FUNCTION_BLOCK fbModTCP_Core IMPLEMENTS iModbusTcpCore
VAR_INPUT
	stTimeStruct : stAircomTimeStruct;																						// Time struct for data ack
END_VAR
VAR_OUTPUT
END_VAR
VAR
	fbModbusTCP 					: FB_MBReadWriteRegs;																	// Main function for ModbusTCP
	arCommQue						: ARRAY[0..GVL_ModbusTCP_Constants.iQueLimit] OF stModTcpQue;							// Que for core
	arModTcpCommandHist				: ARRAY[0..GVL_ModbusTCP_Constants.iCommuniactionHistoryLimit]  OF stModTcpHist;		// Saving of prcesed command
	iWorkStep						: INT;																					// Workstep
	stCommToPerform					: stModTcpQue;																			// Block for process purpose
	iLastQue						: UINT;																					// Que for commands
	iActualQue						: UINT;																					// Actualy performed register of que
	iHistory						: UINT;																					// History record
	rCommunicationTime				: REAL;																					// Time of communication
	fbCommTimeON					: R_TRIG;																				// Start of modbus block - Rise Edge
	fbCommTimeOFF					: F_TRIG;																				// End of modbus block - Falling Edge
	fbErrorDetect					: R_TRIG;																				// Error detected status
	iErrorCalc						: INT;																					// Calculation of errors
	//Visu
	stHMI							: stModTcpCore_HmiData;																	// Data for HMI purpose
	rTimeForStatistic				: REAL;																					// Time variable for statistic calculation - per second
	iLastQueStat					: UINT;																					// Amount of data saved to que
	iActualQueStat					: UINT;																					// Amount od data procesed
	arVisuHist						: ARRAY[0..GVL_ModbusTCP_Constants.iCommuniactionHistoryLimit] OF STRING;				// Command History
	iAmoutOfPerformedCommunications	: DWORD;																				// Sum amount of performed data exchange - per second
	iAmoutOfErrors					: DWORD;																				// Sum amount of errsrs during data exchange - per second
	rTimeforMinuteStatitic			: REAL;																					// Time variable for statistic calculation - per minute
	iLastQueStatMinute				: UINT;																					// Sum amount of performed data exchange - per minute
	iActualQueStatMinute			: UINT;																					// Sum amount of errors during data exchange - per minute
	arErrorHistory					: ARRAY[0..GVL_ModbusTCP_Constants.iCommunicationErrorHistory] OF STRING;				// Data of errors during communicaiotn
	iErrorHistoryIdentifier			: UINT;																					// Calculation of error history
END_VAR

//Rdzeń komuniakcji ModbusTCP
//TO-DO
//Dodać możliwość node - wiele jednoczesnych pracesów
//Dodać możliwosć wymiany inforamcji w Coilach
//Poprawiać ewentualnie wystepujące błędy


ACT_Background();
//Main loop

CASE iWorkStep OF
	0: 		//Inicialization - Step 1
		iWorkStep := 5;

	5: 		//Inicialization - Step 2
		iWorkStep := 10;

	10: 	//Wait for next operaiton
		IF arCommQue[iActualQue].sMachineIndifiner <> '' AND NOT fbModbusTCP.bBusy THEN
			iWorkStep := 15;
		ELSIF NOT fbModbusTCP.bBusy THEN
			IF iActualQue >= GVL_ModbusTCP_Constants.iQueLimit-1 THEN
				iActualQue := 0;
			ELSE
				iActualQue := iActualQue + 1;
			END_IF
		END_IF
	15:		// Check next command
			iWorkStep := 20;
	20:		// Operation prepare - Rewrite for command to perform
		stCommToPerform	:= arCommQue[iActualQue];
		iWorkStep := 25;
	25:		//Clear Que - only one command
		MEMSET(destAddr:=ADR(arCommQue[iActualQue]),fillByte:=0,n:=SIZEOF(stModTcpQue));
		iWorkStep := 30;
		iAmoutOfPerformedCommunications := iAmoutOfPerformedCommunications + 1;
	30:		//Insert command to comm block
		fbModbusTCP.sIPAddr 			:=	stCommToPerform.sIpAdress;
		fbModbusTCP.nUnitID				:=	stCommToPerform.iUnitId;
		fbModbusTCP.nTCPPort			:=	stCommToPerform.iPort;
		fbModbusTCP.nMBReadAddr 		:= 	stCommToPerform.iRegisterReadStartAdress;
		fbModbusTCP.nMBWriteAddr 		:= 	stCommToPerform.iRegisterWriteStartAdress;
			// Dodać error w przypadku ilości rejestrów większych od iWriteRegisterLimit/2
		fbModbusTCP.nReadQuantity 		:=	stCommToPerform.wRegistersReadQuantity;
		fbModbusTCP.nWriteQuantity		:=	stCommToPerform.wRegistersWriteQuantity;
			//Source - Data tobe written in slave | Destination - Data to be read form slave
		fbModbusTCP.cbSrcLength 		:= SIZEOF(stCommToPerform.arRegisterWriteArray^);
		fbModbusTCP.pSrcAddr 			:= stCommToPerform.arRegisterWriteArray;
		fbModbusTCP.cbDestLength 		:= SIZEOF(stCommToPerform.arRegisterReadArray^);
		fbModbusTCP.pDestAddr 			:= stCommToPerform.arRegisterReadArray;
			//Check if history buffer is full - if yes start form 0
		IF iHistory >= GVL_ModbusTCP_Constants.iCommuniactionHistoryLimit THEN
			iHistory := 0;
		END_IF
		arModTcpCommandHist[iHistory].sIpAdress 			:= 	stCommToPerform.sIpAdress;
		arModTcpCommandHist[iHistory].iUnitId 				:=	stCommToPerform.iUnitId;
		arModTcpCommandHist[iHistory].iPort 				:=	stCommToPerform.iPort;
		arModTcpCommandHist[iHistory].sMachineIndifiner 	:= 	stCommToPerform.sMachineIndifiner;
		arModTcpCommandHist[iHistory].sTimeString 			:= 	stTimeStruct.sTimeString;
		arVisuHist[iHistory] := CONCAT(STR1:=arModTcpCommandHist[iHistory].sIpAdress ,STR2:=' | ');
		arVisuHist[iHistory] := CONCAT(STR1:=arVisuHist[iHistory] ,STR2:=arModTcpCommandHist[iHistory].sMachineIndifiner);
		arVisuHist[iHistory] := CONCAT(STR1:=arVisuHist[iHistory] ,STR2:=' | ');
		arVisuHist[iHistory] := CONCAT(STR1:=arVisuHist[iHistory] ,STR2:= arModTcpCommandHist[iHistory].sTimeString);
		arVisuHist[iHistory] := CONCAT(STR1:=arVisuHist[iHistory] ,STR2:=' | ');
		
		iWorkStep := 40;
	40:		// Data exchange start
		fbModbusTCP.bExecute := TRUE;
		IF fbModbusTCP.bBusy THEN
			fbModbusTCP.bExecute := FALSE;
			iWorkStep := 50;
		END_IF
	50: 	//Wait for not busy
		IF NOT fbModbusTCP.bBusy THEN
			iWorkStep := 10;
		END_IF

END_CASE

ACTION ACT_Background:
// Main function
fbModbusTCP();
//Error counting
fbErrorDetect(CLK:= fbModbusTCP.bError);
IF fbErrorDetect.Q THEN
	iErrorCalc := iErrorCalc + 1;
	iAmoutOfErrors := iAmoutOfErrors + 1;
	arErrorHistory[iErrorHistoryIdentifier] := CONCAT(STR1:= stCommToPerform.sMachineIndifiner,STR2:=' | ');
	arErrorHistory[iErrorHistoryIdentifier] := CONCAT(STR1:= arErrorHistory[iErrorHistoryIdentifier],STR2:=stCommToPerform.sIpAdress);
	arErrorHistory[iErrorHistoryIdentifier] := CONCAT(STR1:= arErrorHistory[iErrorHistoryIdentifier],STR2:=' | ');
	arErrorHistory[iErrorHistoryIdentifier] := CONCAT(STR1:= arErrorHistory[iErrorHistoryIdentifier],STR2:=LREAL_TO_FMTSTR(in:=rCommunicationTime,iPrecision:=3,bRound:= FALSE));
	arErrorHistory[iErrorHistoryIdentifier] := CONCAT(STR1:= arErrorHistory[iErrorHistoryIdentifier],STR2:=' | ');
	arErrorHistory[iErrorHistoryIdentifier] := CONCAT(STR1:= arErrorHistory[iErrorHistoryIdentifier],STR2:=UDINT_TO_STRING(fbModbusTCP.nErrId));
	iErrorHistoryIdentifier := iErrorHistoryIdentifier + 1;
END_IF
// Clear amount of errors
IF fbModbusTCP.cbRead <> 0 THEN
	iErrorCalc := 0;
END_IF

//Communication statistic
fbCommTimeON(CLK:= fbModbusTCP.bBusy);
fbCommTimeOFF(CLK:= fbModbusTCP.bBusy);
IF fbCommTimeON.Q THEN
	rCommunicationTime := 0;
END_IF
IF fbModbusTCP.bBusy THEN
	rCommunicationTime := rCommunicationTime + 0.01;
END_IF
IF fbCommTimeOFF.Q THEN
	arModTcpCommandHist[iHistory].rCommandTime := rCommunicationTime;
	arVisuHist[iHistory] := CONCAT(STR1:=arVisuHist[iHistory] ,STR2:=LREAL_TO_FMTSTR(in:=rCommunicationTime,iPrecision:=3,bRound:= FALSE));
	arVisuHist[iHistory] := CONCAT(STR1:=arVisuHist[iHistory] ,STR2:=' | ');
	arModTcpCommandHist[iHistory].nErrorId := fbModbusTCP.nErrId;
	arVisuHist[iHistory] := CONCAT(STR1:=arVisuHist[iHistory] ,STR2:=UDINT_TO_STRING(arModTcpCommandHist[iHistory].nErrorId));
	iHistory := iHistory + 1;
	iActualQueStat := iActualQueStat + 1;
END_IF

//HMI

stHMI.arVisuHist 						:= arVisuHist;
stHMI.arErrorHistory 					:= arErrorHistory;
stHMI.iActualQue 						:= iActualQue;
stHMI.iAmoutOfErrors 					:= iAmoutOfErrors;
stHMI.iAmoutOfPerformedCommunications 	:= iAmoutOfPerformedCommunications;
stHMI.iLastQue 							:= iLastQue;
stHMI.iMessagesPerMinute 				:= iActualQueStatMinute;
stHMI.iPullsPerrMinute					:= iLastQueStatMinute;

IF stHMI.bClearStatistic THEN
	iAmoutOfPerformedCommunications := 0;
	iAmoutOfErrors := 0;
	iActualQueStatMinute := 0;
	iLastQueStatMinute := 0;
	iErrorHistoryIdentifier := 0;
	iHistory := 0;
	stHMI.bClearStatistic := FALSE;
	MEMSET(destAddr:=ADR(arErrorHistory),fillByte:=0,n:= SIZEOF(arErrorHistory));
	MEMSET(destAddr:=ADR(arVisuHist),fillByte:=0,n:= SIZEOF(arVisuHist));
END_IF

IF rTimeForStatistic >= GVL_ModbusTCP_Constants.rTimeForSecondStatistic THEN
	stHMI.iMessagesPerSecond := iActualQueStat;
	stHMI.iPullsPerSecond	:= iLastQueStat;
	iActualQueStatMinute := iActualQueStatMinute + iActualQueStat;
	iLastQueStatMinute	:= iLastQueStatMinute + iLastQueStat;
	iLastQueStat 	:= 0;
	iActualQueStat	:= 0;
	rTimeForStatistic := 0;
END_IF

IF rTimeforMinuteStatitic >= GVL_ModbusTCP_Constants.rTimeForMinuteStatistic THEN
	iActualQueStatMinute := 0;
	iLastQueStatMinute := 0;
	rTimeforMinuteStatitic := 0;
END_IF

rTimeForStatistic := rTimeForStatistic + 0.01;
rTimeforMinuteStatitic := rTimeforMinuteStatitic + 0.01;

fbModbusTCP.tTimeout := GVL_ModbusTCP_Constants.tModbusCommunicationTimeOut;
END_ACTION

METHOD mAddToQue : nModbusTCP_CommandStatus;
VAR_INPUT
	stCommParams	: stModTcpQue;
END_VAR
VAR
END_VAR
IF stCommParams.sIpAdress <> '' AND stCommParams.iPort <> 0 AND stCommParams.sMachineIndifiner <> '' 
AND stCommParams.arRegisterReadArray <> 0 AND stCommParams.arRegisterWriteArray <> 0 AND stCommParams.wRegistersReadQuantity <> 0 AND stCommParams.wRegistersWriteQuantity <> 0
AND stCommParams.wRegistersReadQuantity <= 2*SIZEOF(stCommParams.arRegisterReadArray^) AND stCommParams.wRegistersWriteQuantity <= 2*SIZEOF(stCommParams.arRegisterWriteArray^) THEN
	//IF arCommQue[iLastQue].sMachineIndifiner = stCommParams.sMachineIndifiner THEN
		//mAddToQue := nModbusTCP_CommandStatus.nCommandAlreadyinQue_03;
	//ELSE
		IF iLastQue >= GVL_ModbusTCP_Constants.iQueLimit THEN
			iLastQue := 0;
		END_IF
		IF arCommQue[iLastQue].sMachineIndifiner <> '' THEN
			mAddToQue := nModbusTCP_CommandStatus.nRecordAllreadyInUse_04;
			iLastQue := iLastQue + 1;
			iLastQueStat := iLastQueStat + 1;
		ELSE
			arCommQue[iLastQue] := stCommParams;
			mAddToQue := nModbusTCP_CommandStatus.nCommandPerformed_01;
			iLastQue := iLastQue + 1;
			iLastQueStat := iLastQueStat + 1;
		END_IF
	//END_IF
ELSE
	mAddToQue := nModbusTCP_CommandStatus.nCommandWrongParams_02;
END_IF
END_METHOD

{attribute 'monitoring' := 'call'}
PROPERTY pError : BOOL
GET
pError := iErrorCalc >= GVL_ModbusTCP_Constants.iErrorLimit;
END_GET
END_PROPERTY

END_FUNCTION_BLOCK

(* stored: Version 1.1.0.1, ProductVersion 3.1.4024.13
   POU fbModTCP_Core: Id {1eebaeb0-68d5-4ffe-85ae-e4bdd94758f4}, SpecialFunc None
   Action ACT_Background: Id {3293cfc1-0622-4dd3-8ae2-5d0eb1a0ab74}
   Method mAddToQue: Id {6fcee0ac-971a-4c86-9aba-3116f2e46b99}
   Property pError: Id {362ccfd9-47cc-416e-ab04-599a1a60cbea}
   Get Get: Id {fbab18ed-4e0e-4244-9bec-484473e8833a} *)
